{attribute 'linkalways'} 
{attribute 'no_explicit_call' := 'This FB is a CLASS and must be accessed using methods or properties'}
{attribute 'enable_dynamic_creation'}
FUNCTION_BLOCK _ETcVnInitializableFunction EXTENDS EnumDatatypeBase
VAR
	localData : ETcVnInitializableFunction;
	activeData : REFERENCE TO ETcVnInitializableFunction;
	enumBaseDatatype : _DINT(localData);
END_VAR

METHOD PRIVATE AddLocalEnumeration
VAR_INPUT
	Enumeration : T_MAXSTRING;
	Value : ETcVnInitializableFunction;
END_VAR
AddEnumeration(Enumeration, Value);
END_METHOD

PROPERTY PUBLIC Address : PVOID
GET
Address := ADR(activeData);
END_GET
END_PROPERTY

METHOD PUBLIC ClearReference
VAR_INPUT
END_VAR
activeData REF= localData;
SetBaseDatatypeReference();
END_METHOD

METHOD PUBLIC Clone : I_Datatype
VAR
    pClone : POINTER TO _ETcVnInitializableFunction;
END_VAR
pClone := __NEW(_ETcVnInitializableFunction(InitialValue := Value));
Clone := pClone^;
END_METHOD

METHOD FB_init : BOOL
VAR_INPUT
	bInitRetains : BOOL; // if TRUE, the retain variables are initialized (warm start / cold start)
	bInCopyCode : BOOL;  // if TRUE, the instance afterwards gets moved into the copy code (online change)
	InitialValue : ETcVnInitializableFunction;
END_VAR
localData := InitialValue;
AddBaseDatatype(enumBaseDatatype);
ClearReference();

AddLocalEnumeration('TCVN_IF_OCR', ETcVnInitializableFunction.TCVN_IF_OCR);
END_METHOD

PROPERTY PUBLIC Identifier : T_MAXSTRING
GET
Identifier := 'ETcVnInitializableFunction';
END_GET
END_PROPERTY

METHOD IsEnumeratorValueEqual : BOOL
VAR_INPUT
	Enumerator : I_KeyValueForwardEnumerator;
END_VAR
VAR
	storedValue : ETcVnInitializableFunction;
END_VAR
IF NOT Enumerator.TryGet(storedValue) THEN
	RETURN;
END_IF

IsEnumeratorValueEqual := storedValue = activeData;
END_METHOD

METHOD PUBLIC MakeReferenceTo
VAR_INPUT
	ReferenceTarget : REFERENCE TO ETcVnInitializableFunction;
END_VAR
activeData REF= ReferenceTarget;
SetBaseDatatypeReference();
END_METHOD

METHOD PROTECTED SetBaseDatatypeReference
VAR_INPUT
END_VAR
enumBaseDatatype.MakeReferenceTo(activeData);
END_METHOD

PROPERTY PUBLIC Size : UDINT
GET
Size := SIZEOF(activeData);
END_GET
END_PROPERTY

METHOD TryMakeReferenceTo : BOOL
VAR_INPUT
	Target : I_Datatype;
END_VAR
VAR
	targetAsEnum : I_EnumDatatype;
	pTargetData : POINTER TO ETcVnInitializableFunction;
END_VAR
IF NOT Target.TryResolveAsEnumDatatype(targetAsEnum) THEN
	RETURN;
END_IF

IF targetAsEnum.Identifier <> Identifier THEN
	RETURN;
END_IF

pTargetData := Target.Address;
activeData REF= pTargetData^;
SetBaseDatatypeReference();
TryMakeReferenceTo := TRUE;
END_METHOD

PROPERTY PUBLIC Value : ETcVnInitializableFunction
GET
Value := activeData;
END_GET
SET
activeData := Value;
END_SET
END_PROPERTY

END_FUNCTION_BLOCK

(* stored: Version 1.1.0.1, ProductVersion 3.1.4024.13
   POU _ETcVnInitializableFunction: Id {1c25d15d-5e1b-0412-16ce-c09ec7d2ff9e}, SpecialFunc None
   Folder Core: Id {36122fdf-6bf0-071d-20bb-3f4c1074f2ce}
   Folder Protected: Id {9cc5bb3b-c2d2-08c0-075b-c64a805e1a24}
   Folder Customize: Id {d37dedf2-4975-0ebd-0ae4-97d0b20502d3}
   Folder Constructor: Id {f8d4f82a-e848-0fc7-1f33-62310a95bd67}
   Folder Private: Id {454f0448-f561-0b72-32c9-89319387ee9d}
   Folder Protected: Id {a1d65dca-72a3-0d0f-0249-9e8ce9d71a9e}
   Method AddLocalEnumeration: Id {9eaef364-2774-069d-259a-0166f63cdd54}
   Property Address: Id {ace775b2-3ffc-0429-3d3b-40c62d9e5628}
   Get Get: Id {a41334c4-a0ee-0335-1529-2da64df4cda8}
   Method ClearReference: Id {1e3c2091-6b1d-005e-34f7-c09a13fc1814}
   Method Clone: Id {f8d57376-fda9-038a-3b9a-8d7516c1037e}
   Method FB_init: Id {16f1b62a-05ae-0699-2c02-cdbb8ab3c8af}
   Property Identifier: Id {01e81bde-a89e-0b40-0791-ad5b20728d93}
   Get Get: Id {48fdd895-f914-09b6-00e4-07eac2ea0006}
   Method IsEnumeratorValueEqual: Id {e5f01c09-f87b-0a7b-192a-34fb29fd13ce}
   Method MakeReferenceTo: Id {3d39a30b-d075-0773-2bb8-7443435f6550}
   Method SetBaseDatatypeReference: Id {2ed25592-3fce-000b-366b-33ab4c1e2063}
   Property Size: Id {5a1adbae-2be8-048c-157e-6e1850e401da}
   Get Get: Id {3753d3ca-142f-048a-1cc9-9f283956ff6f}
   Method TryMakeReferenceTo: Id {af116ddf-1f74-07a9-2243-1f8ad8e4bd90}
   Property Value: Id {c140e6ed-b6dc-0745-1563-c1f03018e6fd}
   Get Get: Id {d9de72ae-257d-0aee-0e78-b1f8da48e2bd}
   Set Set: Id {9a48d5a8-7246-0e9e-39dc-7fb1651a790b} *)
